FUNCTION_BLOCK FB_Placing_v2
VAR_INPUT
	Inp_Enable				: BOOL;
	Inp_Reset				: BOOL;
	Inp_SensorBack			: BOOL;
	Inp_SensorMiddle		: BOOL;
	Inp_SensorFront			: BOOL;
	Cmd_Flushing			: BOOL;
	bRobotMove				: BOOL;
	Inp_Done_Place			: BOOL;
	Inp_Req					: BOOL;
	i_Data					: UINT;
	i_Pattern				: UINT;
	i_MaxStacking			: UINT;
	Inp_FB					: BOOL;
	Set_Tmr_Check			: TIME;
	Inp_GlobalReset			: BOOL;
	Inp_ResetData			: BOOL;
	bBypassFGHS				: BOOL;
	CreateID				: STRING;
	
END_VAR
VAR_OUTPUT
	Out_Motor_Fwd			: BOOL;
	Out_Motor_Rev			: BOOL;
	Out_Req					: BOOL;
	Out_FB					: BOOL;
	Out_PalletJammed		: BOOL;
	Out_Rob_Placing			: BOOL;
	CurrentJob				: STRING;
	SeqIndex				: INT;
	PalletOut				: BOOL;
END_VAR
VAR_OUTPUT PERSISTENT
	PalletID				: STRING;
	CounterBarcode			: BYTE;
END_VAR

VAR
	Sts_Flushing			: BOOL;
	o_MaxCycle				: UINT;
	DataTimer				: TON;
	TWatchDog				: TON;
	Sequence				: INT;
END_VAR

VAR_IN_OUT
	AccFlushing				: BYTE;
	Data_Count_Place		: USINT;
	Data_Count_Real			: USINT;
	Data_Incomplete			: UINT;
	Data_Pallet_Total		: UINT;
	Data_Count_Total		: UINT;
END_VAR

(IF Inp_Reset AND Out_PalletJammed THEN // Jika sinyal reset aktif dan palet terjammed
	Out_PalletJammed	:= FALSE; // Matikan sinyal palet terjammed
	Sequence 			:= 0; // Set urutan langkah ke 0
END_IF

IF Inp_Enable THEN // Jika sinyal enable aktif
	
	IF Cmd_Flushing THEN // Jika perintah flushing aktif
		Sts_Flushing:=TRUE; // Set status flushing menjadi TRUE
	END_IF;
	
    CASE Sequence OF // Pilih langkah berdasarkan urutan langkah
        0:	(* Check Motor *) // Langkah 0: Periksa motor
			 Out_Motor_Fwd := TRUE; // Nyalakan motor maju
			 DataTimer(IN:=TRUE, PT:=T#4S); // Mulai timer data dengan durasi 4 detik
			 IF DataTimer.Q OR AccFlushing = 2 THEN // Jika timer data berakhir atau akumulator flushing = 2
				 DataTimer(IN:=FALSE); // Matikan timer data
				 Out_Motor_Fwd	:= FALSE; // Matikan motor maju
				 Sequence		:= 10; // Pergi ke langkah 10
			 END_IF

		10:  (* Check Sensor *) // Langkah 10: Periksa sensor
			CurrentJob		:= 'Check Sensor'; // Tentukan pekerjaan saat ini
			IF (Inp_SensorFront OR Inp_SensorMiddle OR Inp_SensorBack) AND AccFlushing = 2 THEN // Jika salah satu sensor terdeteksi dan akumulator flushing = 2
				Sequence := 600; // Pergi ke langkah 600
			ELSIF (Inp_SensorFront OR Inp_SensorMiddle OR Inp_SensorBack) AND ((Data_Count_Place > o_MaxCycle AND o_MaxCycle <> 0)  OR Sts_Flushing) THEN // Jika salah satu sensor terdeteksi dan jumlah data tempat melebihi siklus maksimum atau status flushing aktif
                Sequence := 500; // Pergi ke langkah 500
            ELSIF Inp_SensorFront THEN // Jika hanya sensor depan terdeteksi
                Sequence := 300; // Pergi ke langkah 300
            ELSIF NOT Inp_SensorFront AND (Inp_SensorMiddle OR Inp_SensorBack)  THEN // Jika tidak ada sensor depan dan salah satu sensor tengah atau belakang terdeteksi
                Sequence := 200; // Pergi ke langkah 200
            ELSE // Jika tidak ada sensor terdeteksi
                Sequence := 100; // Pergi ke langkah 100
            END_IF;
			
			
        100:    (* Request *) // Langkah 100: Kirim permintaan palet
			CurrentJob		:= 'Request Pallet'; // Tentukan pekerjaan saat ini
			Sts_Flushing	:= FALSE; // Matikan status flushing
            Out_Req			:= TRUE; // Aktifkan sinyal permintaan
			Out_FB			:= FALSE; // Matikan sinyal kembali
            IF Inp_FB THEN // Jika sinyal kembali aktif
				DataTimer(IN:=FALSE); // Matikan timer data
                Sequence := 200; // Pergi ke langkah 200
            END_IF;       
			
        200:    (* Pallet Masuk *) // Langkah 200: Palet masuk
			CurrentJob	:= 'Pallet In'; // Tentukan pekerjaan saat ini
			PalletOut	:= FALSE; // Set status keluarnya palet menjadi FALSE
			IF NOT Inp_SensorFront AND NOT Inp_SensorMiddle AND NOT Inp_SensorBack THEN // Jika tidak ada sensor terdeteksi
            	Out_Req := TRUE; // Aktifkan sinyal permintaan
			END_IF
            Out_Motor_Fwd := TRUE; // Nyalakan motor maju
            IF Inp_SensorFront AND (Inp_SensorBack OR Inp_SensorMiddle)  THEN // Jika sensor depan terdeteksi dan salah satu sensor tengah atau belakang terdeteksi
				DataTimer(IN := TRUE,PT := Set_Tmr_Check); // Mulai timer data dengan durasi yang ditentukan
                IF DataTimer.Q THEN // Jika timer data berakhir
					TWatchDog(IN := FALSE); // Matikan watchdog
                    DataTimer(IN:=FALSE); // Matikan timer data
					Out_PalletJammed	:= FALSE; // Matikan sinyal palet terjammed
					Out_Motor_Fwd		:= FALSE; // Matikan motor maju
           			Out_Req				:= FALSE; // Matikan sinyal permintaan
                    Sequence			:= 300; // Pergi ke langkah 300
                END_IF;    
			ELSE
				TWatchDog(IN := TRUE, PT := T#15S); // Mulai watchdog dengan durasi 15 detik
				IF TWatchDog.Q THEN // Jika watchdog berakhir
					Sequence	:= 9999; // Pergi ke langkah 9999
				END_IF;
            END_IF;
			
        300: // Langkah 300: Periksa siklus
			CurrentJob	:= 'Check Cycle'; // Tentukan pekerjaan saat ini
			IF o_MaxCycle <> 0 THEN // Jika siklus maksimum tidak sama dengan 0
				IF o_MaxCycle >= Data_Count_Place  THEN // Jika siklus maksimum lebih besar atau sama dengan jumlah data tempat
					Sequence := 400; // Pergi ke langkah 400
				ELSE
					DataTimer(IN := TRUE,PT := T#2S); // Mulai timer data dengan durasi 2 detik
					IF DataTimer.Q THEN // Jika timer data berakhir
						DataTimer(IN:=FALSE); // Matikan timer data
						Sequence := 500; // Pergi ke langkah 500
					END_IF;
				END_IF;
			END_IF
			
        400: // Langkah 400: Tempat siap
			CurrentJob		:= 'Place Ready'; // Tentukan pekerjaan saat ini
			AccFlushing		:= 0; // Set akumulator flushing menjadi 0
            Out_Rob_Placing := TRUE; // Aktifkan sinyal robot meletakkan
			PalletID			:= CreateID; // Tentukan ID palet
            IF Inp_Done_Place THEN // Jika proses penempatan selesai
                    Data_Count_Real		:= Data_Count_Real + 1; // Tambahkan jumlah data tempat yang sebenarnya
                    Data_Count_Place	:= Data_Count_Place + 1; // Tambahkan jumlah data tempat
                    Sequence 			:= 450; // Pergi ke langkah 450
            ELSIF (Cmd_Flushing OR Sts_Flushing) AND NOT bRobotMove THEN // Jika perintah flushing atau status flushing aktif dan robot tidak bergerak
                Data_Incomplete			:= Data_Incomplete + 1; // Tambahkan jumlah data yang tidak lengkap
                Sts_Flushing			:= TRUE; // Set status flushing menjadi TRUE
                Sequence 				:= 500; // Pergi ke langkah 500				
            END_IF;
			
        450: // Langkah 450: Persiapan tempat selesai
            Out_Rob_Placing := FALSE; // Matikan sinyal robot meletakkan
            IF NOT Inp_Done_Place THEN // Jika proses penempatan belum selesai
                Sequence := 460; // Pergi ke langkah 460
            END_IF;	
			
		460: // Langkah 460: Penyelesaian penempatan
			IF PalletID <> '' THEN // Jika ID palet tidak kosong
				CounterBarcode	:= Data_Count_Real; // Tentukan counter barcode
				Sequence 		:= 300; // Pergi ke langkah 300
			END_IF
			
		500: // Langkah 500: Buat ID palet
			CurrentJob		:= 'Create Pallet ID'; // Tentukan pekerjaan saat ini
			DataTimer(IN := TRUE,PT := T#500MS); // Mulai timer data dengan durasi 500 ms
			IF DataTimer.Q THEN // Jika timer data berakhir
				DataTimer(IN := FALSE); // Matikan timer data
				Sequence		:= 550; // Pergi ke langkah 550
			END_IF
						
		550: // Langkah 550: Selesai pembuatan ID palet
			AccFlushing		:= 1; // Set akumulator flushing menjadi 1
			Sequence		:= 600; // Pergi ke langkah 600
			
		600: // Langkah 600: Menunggu akumulator flushing
			Out_Rob_Placing := FALSE; // Matikan sinyal robot meletakkan
			Out_FB 			:= FALSE; // Matikan sinyal kembali
			Out_Req 		:= FALSE; // Matikan sinyal permintaan
			CurrentJob		:= 'Waiting Acc Flushing'; // Tentukan pekerjaan saat ini
			IF (PalletID <> '' AND AccFlushing = 2) OR bBypassFGHS OR Data_Count_Real = 0 THEN // Jika ID palet tidak kosong dan akumulator flushing = 2 atau bypass FGHS aktif atau jumlah data tempat sebenarnya = 0
                Sequence := 900; // Pergi ke langkah 900
            END_IF;
		
		900:	(* Positioning Pallet Out *) // Langkah 900: Posisi palet keluar
			CurrentJob		:= 'Positioning Pallet Out'; // Tentukan pekerjaan saat ini
			Out_Rob_Placing := FALSE; // Matikan sinyal robot meletakkan
			Out_FB 			:= TRUE; // Aktifkan sinyal kembali
			Out_Req 		:= TRUE; // Aktifkan sinyal permintaan
			Out_Motor_Rev	:= TRUE; // Nyalakan motor mundur
            IF Inp_SensorBack THEN // Jika sensor belakang terdeteksi
                DataTimer(IN := TRUE,PT := T#100MS); // Mulai timer data dengan durasi 100 ms
                IF DataTimer.Q THEN // Jika timer data berakhir
					TWatchDog(IN := FALSE); // Matikan watchdog
					DataTimer(IN:=FALSE); // Matikan timer data
					Out_Motor_Rev	:= FALSE; // Matikan motor mundur
                    Sequence		:= 1000; // Pergi ke langkah 1000
                END_IF;
			ELSE
				TWatchDog(IN := TRUE, PT := T#15S); // Mulai watchdog dengan durasi 15 detik
				IF TWatchDog.Q THEN // Jika watchdog berakhir
					Sequence		:= 9999; // Pergi ke langkah 9999
				END_IF;
            END_IF;
			            
        1000:    (* Menunggu Request *) // Langkah 1000: Menunggu permintaan
			Out_Rob_Placing := FALSE; // Matikan sinyal robot meletakkan
			CurrentJob		:= 'Waiting Request'; // Tentukan pekerjaan saat ini
			Out_FB 			:= TRUE; // Aktifkan sinyal kembali
			Out_Req 		:= TRUE; // Aktifkan sinyal permintaan
            IF Inp_Req AND Inp_FB AND (AccFlushing = 2 OR bBypassFGHS OR Data_Count_Real = 0) THEN // Jika permintaan dan sinyal kembali aktif dan akumulator flushing = 2 atau bypass FGHS aktif atau jumlah data tempat sebenarnya = 0
                Sequence := 1100; // Pergi ke langkah 1100
            END_IF;
			
        1100:    (* Pallet Keluar *) // Langkah 1100: Palet keluar
			CurrentJob		:= 'Pallet Out'; // Tentukan pekerjaan saat ini
            Out_Motor_Rev	:= TRUE; // Nyalakan motor mundur
            IF (NOT Inp_SensorBack AND NOT Inp_SensorFront )AND NOT Inp_Req THEN // Jika tidak ada sensor depan dan belakang dan tidak ada permintaan
                DataTimer(IN := TRUE,PT := T#500ms); // Mulai timer data dengan durasi 500 ms
                IF DataTimer.Q THEN // Jika timer data berakhir
					TWatchDog(IN := FALSE); // Matikan watchdog
					DataTimer(IN:=FALSE); // Matikan timer data
					Out_FB			:= FALSE; // Matikan sinyal kembali
					Out_Motor_Rev	:= FALSE; // Matikan motor mundur
                    Sequence		:= 1200; // Pergi ke langkah 1200
                END_IF;
			ELSE
				TWatchDog(IN := TRUE, PT := T#15S); // Mulai watchdog dengan durasi 15 detik
				IF TWatchDog.Q THEN // Jika watchdog berakhir
					Sequence		:= 9999; // Pergi ke langkah 9999
				END_IF;
            END_IF;
			
        1200: // Langkah 1200: Selesai palet keluar
			AccFlushing			:= 0; // Set akumulator flushing menjadi 0
			IF NOT Sts_Flushing THEN // Jika status flushing tidak aktif
			Data_Pallet_Total	:= Data_Pallet_Total + 1; // Tambahkan jumlah palet secara total
			END_IF
			Data_Count_Total	:= Data_Count_Total + Data_Count_Real; // Tambahkan jumlah data tempat secara total
			Sequence			:= 1300; // Pergi ke langkah 1300
		   
        1300: // Langkah 1300: Persiapan ulang
			CounterBarcode		:= 0; // Reset counter barcode
            Data_Count_Real		:= 0; // Reset jumlah data tempat sebenarnya
			Data_Count_Place	:= 1; // Reset jumlah data tempat
			PalletID			:= ''; // Reset ID palet
			PalletOut			:= TRUE; // Set status keluar palet menjadi TRUE
            IF NOT Inp_Req THEN // Jika tidak ada permintaan
                Sequence		:= 100; // Pergi ke langkah 100
            END_IF;
			
		9999: // Langkah 9999: Penanganan timeout
			TWatchDog(IN := FALSE); // Matikan watchdog
			DataTimer(IN:=FALSE); // Matikan timer data
			Out_PalletJammed	:= TRUE; // Aktifkan sinyal palet terjammed
			Out_Motor_Rev 		:= FALSE; // Matikan motor mundur
			Out_Motor_Fwd 		:= FALSE; // Matikan motor maju
			
        END_CASE;
ELSE
  	DataTimer(IN:=FALSE); // Matikan timer data
	TWatchDog(IN := FALSE); // Matikan watchdog
	Out_Motor_Rev 		:= FALSE; // Matikan motor mundur
	Out_Motor_Fwd 		:= FALSE; // Matikan motor maju
    Out_Rob_Placing 	:= FALSE; // Matikan sinyal robot meletakkan
    Out_Req 			:= FALSE; // Matikan sinyal permintaan
	Out_FB 				:= FALSE; // Matikan sinyal kembali
	CurrentJob			:= 'Machine Stopped'; // Tentukan pekerjaan saat ini
	IF Inp_GlobalReset THEN // Jika reset global aktif
        Sequence 		:= 0; // Set urutan langkah ke 0
        Out_FB 			:= FALSE; // Matikan sinyal kembali
        Sts_Flushing 	:= FALSE; // Matikan status flushing
    END_IF;
END_IF;

//Sequence Index
SeqIndex	:= Sequence; // Set indeks urutan langkah

IF Data_Count_Place = 0 THEN // Jika jumlah data tempat = 0
    Data_Count_Place  := 1; // Set jumlah data tempat menjadi 1
END_IF;

Data_Count_Place := Data_Count_Real+1; // Tentukan jumlah data tempat dengan menambahkan jumlah data tempat sebenarnya dengan 1

// Calculate Max Cycle
o_MaxCycle :=i_Data*i_MaxStacking; // Hitung siklus maksimum

IF Inp_ResetData THEN // Jika reset data aktif
    Data_Count_Total	:= 0; // Reset jumlah data tempat secara total
    Data_Pallet_Total 	:= 0; // Reset jumlah palet secara total
    Data_Incomplete 	:= 0; // Reset jumlah data yang tidak lengkap
END_IF;

END_FUNCTION_BLOCK

(* stored: Version 1.1.0.1, ProductVersion 3.1.4024.6
   POU FB_Placing_v2: Id {773ff4c9-68b5-407a-bcdf-4f8ead4c792f}, SpecialFunc None *)
